(* PLC project Senza_nome, Sconosciuto Senza_nome 1 *)
(* stored: creationDateTime 2026-08-26T12:54:19, modificationDateTime 2026-08-26T14:44:57 *)

PROGRAM program0
  VAR
    I_Cucina : BOOL;
    I_Cucina0 : BOOL;
    I_Camera : BOOL;
    I_Sogiorno : BOOL;
    I_Sogiorno0 : BOOL;
    I_Bagno : BOOL;
    I_Dormitorio1 : BOOL;
    I_Dormitorio2 : BOOL;
    I_Dormitorio3 : BOOL;
    P_Salita : BOOL;
    P_Discesa : BOOL;
    P_Stop : BOOL;
    FC_Alto : BOOL;
    FC_Basso : BOOL;
    I_Chiave : BOOL;
    FC_Aperto : BOOL;
    FC_Chiuso : BOOL;
    Fotocellula : BOOL;
    Q_Cucina : BOOL;
    Q_Camera : BOOL;
    Q_Soggiorno : BOOL;
    Q_Bagno : BOOL;
    Q_Dormitorio1 : BOOL;
    Q_Dormitorio2 : BOOL;
    Q_Dormitorio3 : BOOL;
    Q_Discesa : BOOL;
    Q_Salita : BOOL;
    Q_Cancello_Avanti : BOOL;
    Q_Cancello_Indietro : BOOL;
    M_Stato_Cucina : BOOL;
    M_Stato_Camera : BOOL;
    M_Stato_Dormi1 : BOOL;
    M_Stato_Dormi2 : BOOL;
    M_Stato_Dormi3 : BOOL;
    TON0 : TON;
    TON_Q : BOOL;
  END_VAR

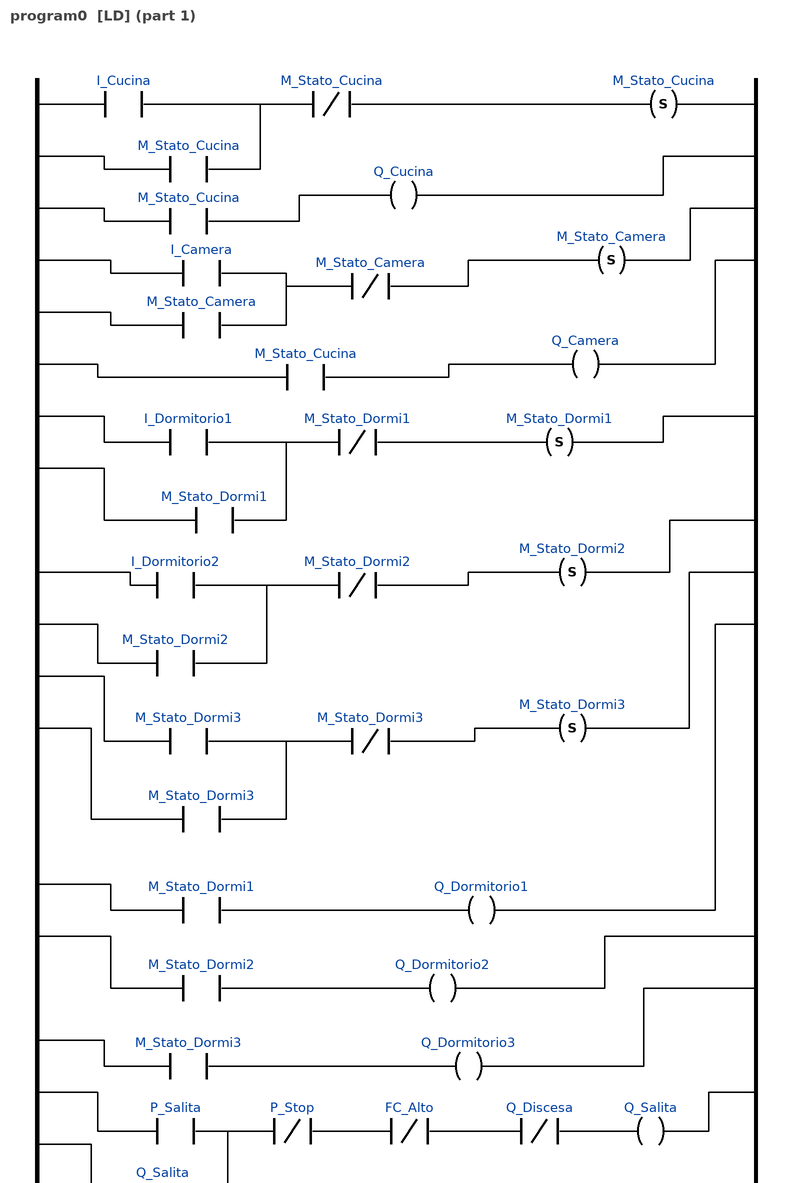
(* LD diagram, written out as Structured Text *)
IF (I_Cucina OR M_Stato_Cucina) AND NOT M_Stato_Cucina THEN M_Stato_Cucina := TRUE; END_IF;
Q_Cucina := M_Stato_Cucina;
IF (I_Camera OR M_Stato_Camera) AND NOT M_Stato_Camera THEN M_Stato_Camera := TRUE; END_IF;
Q_Camera := M_Stato_Cucina;
IF (I_Dormitorio1 OR M_Stato_Dormi1) AND NOT M_Stato_Dormi1 THEN M_Stato_Dormi1 := TRUE; END_IF;
IF (I_Dormitorio2 OR M_Stato_Dormi2) AND NOT M_Stato_Dormi2 THEN M_Stato_Dormi2 := TRUE; END_IF;
IF M_Stato_Dormi3 AND NOT M_Stato_Dormi3 THEN M_Stato_Dormi3 := TRUE; END_IF;
Q_Dormitorio1 := M_Stato_Dormi1;
Q_Dormitorio2 := M_Stato_Dormi2;
Q_Dormitorio3 := M_Stato_Dormi3;
Q_Salita := (P_Salita OR NOT Q_Salita) AND NOT P_Stop AND NOT FC_Alto AND NOT Q_Discesa;
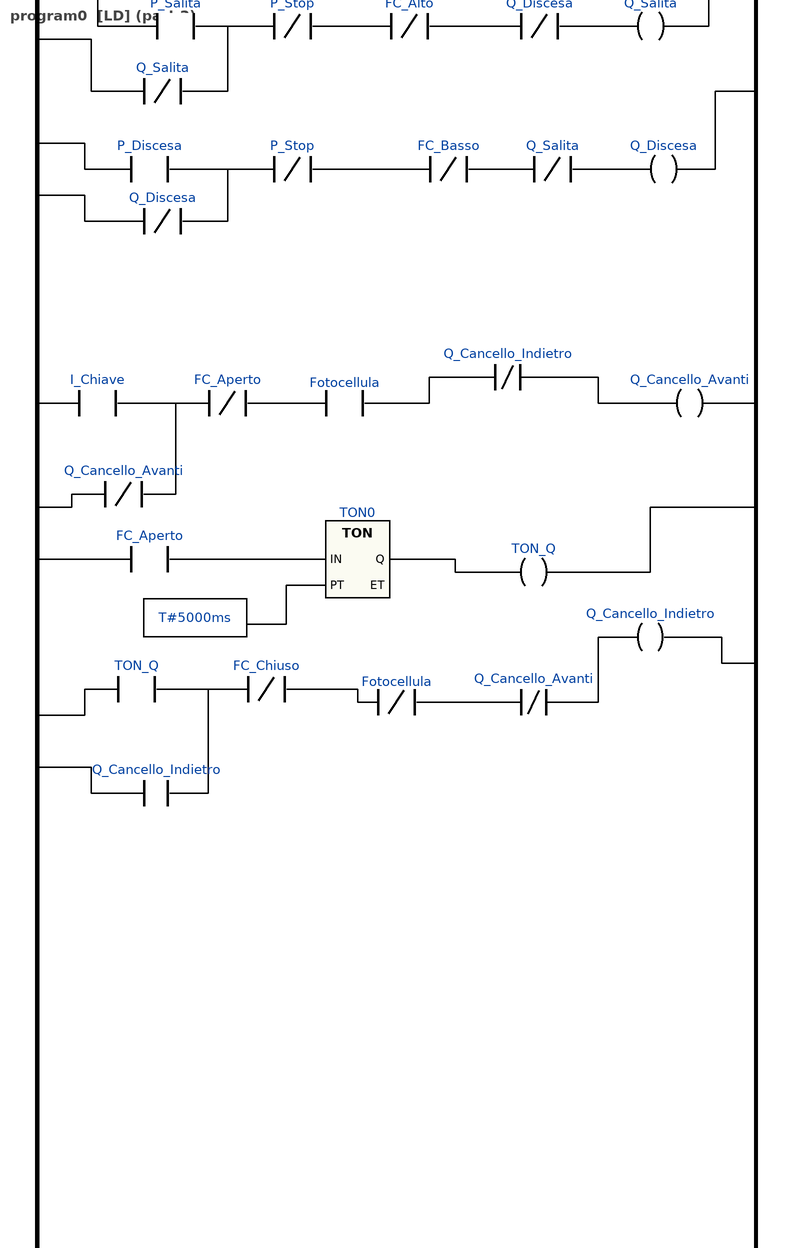
Q_Discesa := (P_Discesa OR NOT Q_Discesa) AND NOT P_Stop AND NOT FC_Basso AND NOT Q_Salita;
Q_Cancello_Avanti := (I_Chiave OR NOT Q_Cancello_Avanti) AND NOT FC_Aperto AND Fotocellula AND NOT Q_Cancello_Indietro;
TON0(IN := FC_Aperto, PT := T#5000ms);
TON_Q := TON0.Q;
Q_Cancello_Indietro := (TON_Q OR Q_Cancello_Indietro) AND NOT FC_Chiuso AND NOT Fotocellula AND NOT Q_Cancello_Avanti;
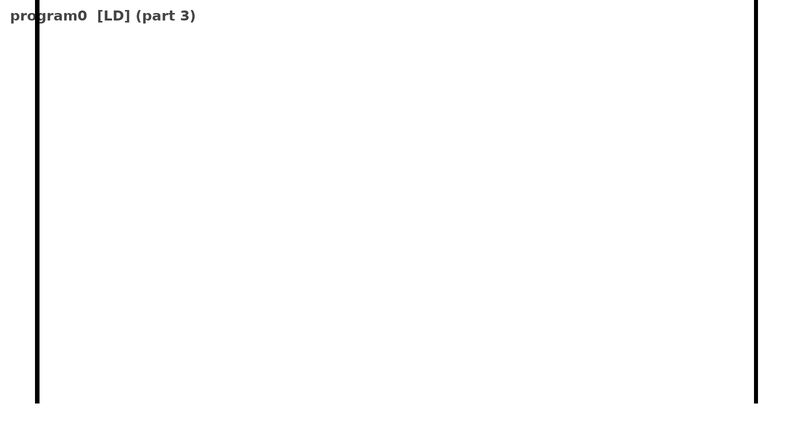
END_PROGRAM

CONFIGURATION Config0
  RESOURCE Res0 ON PLC
    TASK task0(INTERVAL := T#20ms, PRIORITY := 0);
    PROGRAM instance0 WITH task0 : program0;
  END_RESOURCE
END_CONFIGURATION
